// Mitsubishi GX Works2 project: LRI.gx2   PLC: Q03UDV

PROGRAM MAIN
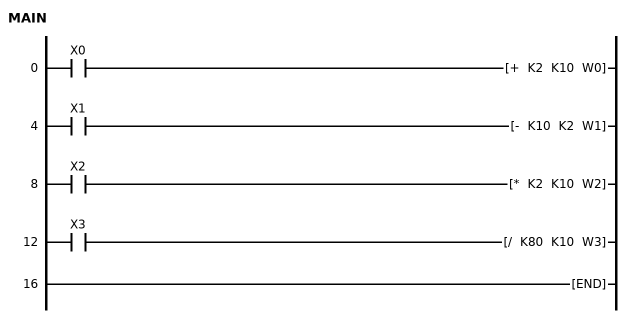
0     LD      X0
      +       K2 K10 W0
4     LD      X1
      -       K10 K2 W1
8     LD      X2
      *       K2 K10 W2
12    LD      X3
      /       K80 K10 W3
16    END
END_PROGRAM
